(* IEC 61131-3 sources: WarwickBoringPLC/, 5 files *)

(* ---- mainGVL.gvl ---- *)
// For main global variables
// **********************************************************************
// ** VERSION 1.0.0 - Aaron 29/01/23**
// The main global variable list
//
// Changelog:
// - Added ME flowmeter
// **********************************************************************

{attribute 'qualified_only'}
VAR_GLOBAL
	// Saftey
;
	// Is inerlocked
	isSystemInterlocked: BOOL; // True when estop or problem occurs, requires reset to clear;
	isResettable: BOOL := FALSE; // True when system can be reset

	isSystemEnabled: BOOL := FALSE; // True when system is running and enabled

	isPoweredOn: BOOL := FALSE; // Power button

	isIssue: BOOL := FALSE; // Is there something causing an issue (causing interlock)

	// General Values
	;
	cpuLoad: UDINT;

	// Material Extraction
	meFlowMeterCount: INT;
	meFlowMeterRate: REAL;

END_VAR

(* ---- mGVL.gvl ---- *)
// This global variable list is to instanitate all of the IO variables to the named variables.
{attribute 'qualified_only'}
VAR_GLOBAL
	// CC E STOP - Switch
	eStopCC: BOOL;
	// HPU relief valve to enable/disable hydraulics
	hpuReliefValve: BOOL;

	// Hydraulic Pressure sensor A
	hydraulicPressureSensorA: INT;

	// Valve Amplifiers
	;
	// Motor Valve Amplifier
	motValveAmp: INT;
	// Thrust Cylinder A Valve Amplifier
	thrAValveAmp: INT;
	// Thrust Cylinder B Valve Amplifier
	thrBValveAmp: INT;
	// Thrust Cylinder C Valve Amplifier
	thrCValveAmp: INT;
	// Thrust Cylinder D Valve Amplifier
	thrDValveAmp: INT;

	// Gripper Amplifiers
	grpAPwrAmp: INT;
	grpBPwrAmp: INT;

	// Gripper A Directions
	grpADirA: BOOL;
	grpADirB: BOOL;

	// Gripper B Directions
	grpBDirA: BOOL;
	grpBDirB: BOOL;
END_VAR

(* ---- visuGVL.gvl ---- *)
// GVL for the visualisations
{attribute 'qualified_only'}
VAR_GLOBAL
	visuEstop: BOOL := FALSE; // UI E Stop, true when pressed

	resetButton : BOOL := FALSE;

	powerSlider: INT := 0; // Power Slider

	extendButton: BOOL := FALSE;
	retractButton: BOOL := FALSE;

	tAEn: BOOL := FALSE;
	tBEn: BOOL := FALSE;
	tCEn: BOOL := FALSE;
	tDEn: BOOL := FALSE;
	motEn: BOOL := FALSE;
	grpAEn: BOOL := FALSE;
	grpBEn: BOOL := FALSE;

END_VAR

(* ---- MaterialExtraction.st ---- *)
PROGRAM MaterialExtraction
VAR
	// Flow meter triggers
	meFlowMeterCountTrigger : R_TRIG; (* to catch the rising signal edge *)
  	meFlowMeterResetTrigger : R_TRIG; (* to catch the rising signal edge *)

	// Flow meter rate calculation
	tDelta, tCurrent, tLast : TIME;
END_VAR

// **********************************************************************
// ** VERSION 1.0.0 - Aaron 29/01/23**
// Carries out Material Extraction logic
//
// Changelog:
// - Added ME flowmeter
// **********************************************************************

meFlowMeterCountTrigger (CLK := mGVL.meFlowMeterPulse); (* finds the counting up events *)
meFlowMeterResetTrigger (CLK := visuGVL.meResetFlowMeter); (* finds the clear commands *)

IF meFlowMeterCountTrigger.Q
THEN
	mainGVL.meFlowMeterCount := mainGVL.meFlowMeterCount + 1;

	tCurrent := TO_TIME(SysTimeGetMs());

	// Calculate delta
	tDelta := tCurrent - tLast; // ms

	// Calculate rate
	mainGVL.meFlowMeterRate := 1000 / TIME_TO_REAL(tDelta); // L per second

	tLast := tCurrent;

END_IF;
IF meFlowMeterResetTrigger.Q
	THEN mainGVL.meFlowMeterCount := 0;
END_IF;

(* ---- VariableMapping.st ---- *)
PROGRAM VariableMapping
VAR
END_VAR

// Map all of the variables to the IO

// Inputs
mGVL.hydraulicPressureSensorA := ACI_3;
mGVL.eStopCC := DI_0;

// Outputs
DO_25 := mGVL.hpuReliefValve;
